{attribute 'linkalways'} 
{attribute 'no_explicit_call' := 'This FB is a CLASS and must be accessed using methods or properties'}
{attribute 'enable_dynamic_creation'}
FUNCTION_BLOCK Node_F_VN_WarpAffine_Point EXTENDS VisionNode
VAR
	aSrcPoint : _TcVnPoint2_LREAL;
    aDestPoint : _TcVnPoint2_LREAL;
    aTransformationMatrix : _TcVnMatrix2x3_LREAL;
    hrPrev : _HRESULT(S_OK);
	hresult : _HRESULT(S_OK);
END_VAR

METHOD PUBLIC  Clone : I_Node
VAR
	pNode : POINTER TO Node_F_VN_WarpAffine_Point;
END_VAR
pNode := __NEW(Node_F_VN_WarpAffine_Point);
Clone := pNode^;
END_METHOD

METHOD FB_init : BOOL
VAR_INPUT
	bInitRetains : BOOL; // if TRUE, the retain variables are initialized (warm start / cold start)
	bInCopyCode : BOOL;  // if TRUE, the instance afterwards gets moved into the copy code (online change)
END_VAR
AddInput('aSrcPoint', aSrcPoint);
AddInput('aTransformationMatrix', aTransformationMatrix);
AddInput('hrPrev', hrPrev);
AddOutput('aDestPoint', aDestPoint);
AddOutput('hresult',hresult);
END_METHOD

METHOD PROTECTED OnExecute
hresult.Value := F_VN_WarpAffine_Point(
	aSrcPoint := aSrcPoint.Value, 
	aDestPoint := aDestPoint.Value, 
	aTransformationMatrix := aTransformationMatrix.Value, 
	hrPrev := hrPrev.Value);
END_METHOD

METHOD PUBLIC PreExecutionCheck
VAR_INPUT
	Check : I_PreExecutionChecks;
END_VAR
END_METHOD

END_FUNCTION_BLOCK

(* stored: Version 1.1.0.1, ProductVersion 3.1.4024.13
   POU Node_F_VN_WarpAffine_Point: Id {ed597c2d-ee29-0e12-1347-f1ba5e41f812}, SpecialFunc None
   Folder Constructor: Id {b6550ad9-470e-0a1d-27d2-5b481edc9c55}
   Method Clone: Id {f05e10ab-e105-0750-0d2e-099610193a7d}
   Method FB_init: Id {2964a44c-c297-04c9-256d-31f61539a661}
   Method OnExecute: Id {92d1e3db-fff7-03d7-3eaa-d27e74c03ba2}
   Method PreExecutionCheck: Id {c83a43ad-a608-0897-1020-e1515f9cc4c9} *)
